// TIA Portal project "TIA_PP" (V19)

(* hardware
DEVICE "HMI_1"  KTP400 Basic PN
   slot 0: "HMI_1"  HMI  6AV2 123-2DB03-0AX0  13.0.1.0
   slot 1: "HMI_RT_1"  KTP400 Basic PN  6AV2 123-2DB03-0AX0  13.0.1.0
   slot 5: "HMI_1.IE_CP_1"  PROFINET Interface
      slot 1: "PROFINET Interface_1"  PROFINET Interface
         slot 1: "Port_1"  Port
DEVICE "S7-1200 station_1"  S7-1200 Station
   slot 0: "Rack_0"  Rack  V1.0
   slot 1: "PLC_1"  CPU 1212C AC/DC/Rly  6ES7 212-1BE40-0XB0  V4.1
*)

// ===== PLC "PLC_1"  CPU 1212C AC/DC/Rly =====

VAR_GLOBAL   // PLC tag table "Default tag table"
   "Tag_1" AT %MD5 : DWord;
   "Tag_2" AT %MD0 : DWord;
   "Tag_4" AT %MW5 : Word;
   "Tag_3" AT %MW10 : Int;
   "Tag_5" AT %M100.0 : Bool;
   "Warning light" AT %Q0.0 : Bool;
   "Tag_7" AT %M100.1 : Bool;
   "Motor1" AT %Q0.1 : Bool;
   "Tag_9" AT %MD5 : Time;
   "Tag_10" AT %MD12 : Real;
   "Tag_11" AT %MW15 : Int;
   "Tag_12" AT %ID30 : DWord;
   "Tag_13" AT %MD22 : Real;
   "Tag_14" AT %MW50 : Word;
   "LED" AT %Q0.2 : Bool;
   "Tag_16" AT %ID34 : DWord;
   "Tag_17" AT %MD25 : Real;
   "Tag_18" AT %MD26 : Real;
   "Fill Valve" AT %QD30 : Real;
   "Drain Valve" AT %QD34 : Real;
   "Tag_19" AT %M200.0 : Bool;
   "Tag_20" AT %M200.1 : Bool;
   "Animation bit" AT %M40.0 : Bool;
   "Clock_Byte" AT %MB300 : Byte;
   "Clock_10Hz" AT %M300.0 : Bool;
   "Clock_5Hz" AT %M300.1 : Bool;
   "Clock_2.5Hz" AT %M300.2 : Bool;
   "Clock_2Hz" AT %M300.3 : Bool;
   "Clock_1.25Hz" AT %M300.4 : Bool;
   "Clock_1Hz" AT %M300.5 : Bool;
   "Clock_0.625Hz" AT %M300.6 : Bool;
   "Clock_0.5Hz" AT %M300.7 : Bool;
   "Tag_21" AT %MB60 : Byte;
   "roller" AT %MD60 : Real;
   "roller_2" AT %MD70 : Real;
   "Tag_22" AT %MD65 : Real;
   "Tag_23" AT %MW60 : Int;
   "Tag_24" AT %MW65 : Int;
   "Down" AT %M90.0 : Bool;
   "Up" AT %M90.1 : Bool;
   "Tag_25" AT %MW75 : Int;
   "Tag_26" AT %MW78 : Int;
   "Tag_27" AT %MW80 : Int;
   "Alarm bit" AT %M99.0 : Bool;
   "Alarm register" AT %MW99 : Int;
   "OK bit" AT %M99.1 : Bool;
   "Reset Alarm" AT %M99.2 : Bool;
   "Start Button" AT %I0.0 : Bool;
   "Tag_28" AT %M0.1 : Bool;
   "Tag_6" AT %M0.2 : Bool;
   "Tag_15" AT %M0.3 : Bool;
   "Elpased time" AT %MD1 : Time;
   "Motor 2" AT %Q0.3 : Bool;
   "Tag_30" AT %Q0.4 : Bool;
   "LED1" AT %Q0.5 : Bool;
   "LED2" AT %Q0.6 : Bool;
   "Manual Button" AT %I0.5 : Bool;
   "Filling Button" AT %I0.6 : Bool;
   "Filling Value" AT %Q0.7 : Bool;
   "Draining Button" AT %I0.7 : Bool;
   "Draining Value" AT %Q1.0 : Bool;
   "Auto Button" AT %I0.1 : Bool;
   "Filling Button(1)" AT %I0.2 : Bool;
   "Tag_8" AT %M0.5 : Bool;
   "Tag_29" AT %M0.7 : Bool;
   "Tag_31" AT %M1.0 : Bool;
   "E-button" AT %M10.0 : Bool;
   "Stop Button" AT %M10.1 : Bool;
END_VAR

// folder: Basic Functions

DATA_BLOCK "PulseGenerator_DB"   // DB2
{ S7_Optimized_Access := 'TRUE' }
VERSION : 0.1
// stored: InstanceOfName PulseGenerator
"PulseGenerator"
BEGIN
END_DATA_BLOCK

DATA_BLOCK "ON-OFF Loop control_DB"   // DB3
{ S7_Optimized_Access := 'TRUE' }
VERSION : 0.1
// stored: InstanceOfName ON-OFF Loop control
"ON-OFF Loop control"
BEGIN
END_DATA_BLOCK

// folder: System blocks/Program resources

DATA_BLOCK "TP"   // DB1
{ S7_Optimized_Access := 'TRUE' }
AUTHOR : Simatic
FAMILY : IEC
NAME : IEC_TMR
VERSION : 1.0
// stored: InstanceOfName IEC_TIMER
"IEC_TIMER"
BEGIN
END_DATA_BLOCK

DATA_BLOCK "IEC_Timer_0_DB"   // DB4
{ S7_Optimized_Access := 'TRUE' }
AUTHOR : Simatic
FAMILY : IEC
NAME : IEC_TMR
VERSION : 1.0
// stored: InstanceOfName IEC_TIMER
"IEC_TIMER"
BEGIN
END_DATA_BLOCK

DATA_BLOCK "IEC_Timer_0_DB_1"   // DB5
{ S7_Optimized_Access := 'TRUE' }
AUTHOR : Simatic
FAMILY : IEC
NAME : IEC_TMR
VERSION : 1.0
// stored: InstanceOfName IEC_TIMER
"IEC_TIMER"
BEGIN
END_DATA_BLOCK

DATA_BLOCK "TON"   // DB6
{ S7_Optimized_Access := 'TRUE' }
AUTHOR : Simatic
FAMILY : IEC
NAME : IEC_TMR
VERSION : 1.0
// stored: InstanceOfName IEC_TIMER
"IEC_TIMER"
BEGIN
END_DATA_BLOCK

DATA_BLOCK "TOFF"   // DB7
{ S7_Optimized_Access := 'TRUE' }
AUTHOR : Simatic
FAMILY : IEC
NAME : IEC_TMR
VERSION : 1.0
// stored: InstanceOfName IEC_TIMER
"IEC_TIMER"
BEGIN
END_DATA_BLOCK

// folder: (top level)

FUNCTION "MHJ-PLC-Lab-Function-S71200" : Void   // FC1, SCL
{ S7_Optimized_Access := 'TRUE' }
VERSION : 0.1
   VAR_TEMP
      rdTimeReturn : Int;
      outputTime : DTL;
      SyncVal : Byte;
      forVal : Int;
      forVal_2 : Int;
      Value : Byte;
   END_VAR
   VAR CONSTANT
      CompVal : Byte := 16#34;
      Value_01 : Byte := 16#11;
      Value_01_DW : DWord := 16#A165_D992;
      Value_02_DW : DWord := 16#58BE_4401;
   END_VAR
BEGIN

   #Value := PEEK(area := 16#82,
                  dbNumber := 0,
                  byteOffset := 511);
   #Value := #Value + 1;

   POKE(area := 16#82,
        dbNumber := 0,
        byteOffset := 511,
        value := #Value);

   POKE(area := 16#81,
        dbNumber := 0,
        byteOffset := 1016,
        value := #Value_01_DW);
   POKE(area := 16#81,
        dbNumber := 0,
        byteOffset := 1020,
        value := #Value_02_DW);

   POKE(area := 16#81,
        dbNumber := 0,
        byteOffset := 511,
        value := B#16#00);

   FOR #forVal := 0 TO 120 DO
       FOR #forVal_2 := 0 TO 10 DO
           #rdTimeReturn := RD_SYS_T(#outputTime);
           #rdTimeReturn := WR_SYS_T(#outputTime);
           #rdTimeReturn := RD_SYS_T(#outputTime);
           #rdTimeReturn := WR_SYS_T(#outputTime);
       END_FOR;
       #SyncVal := PEEK(area := 16#81,
                        dbNumber := 0,
                        byteOffset := 511);
       IF #SyncVal = #CompVal THEN
           GOTO M_1;
       END_IF;
   END_FOR;
   RETURN;

   M_1:
   POKE(area := 16#81,
        dbNumber := 0,
        byteOffset := 511,
        value := B#16#0);
END_FUNCTION

ORGANIZATION_BLOCK "Main"   // OB1, LAD, ProgramCycle
TITLE = "Main Program Sweep (Cycle)"
{ S7_Optimized_Access := 'TRUE' }
VERSION : 0.1
   VAR_INPUT
      Initial_Call : Bool;   // Initial call of this OB
      Remanence : Bool;   // =True, if remanent data are available
   END_VAR
BEGIN

REGION Network 1
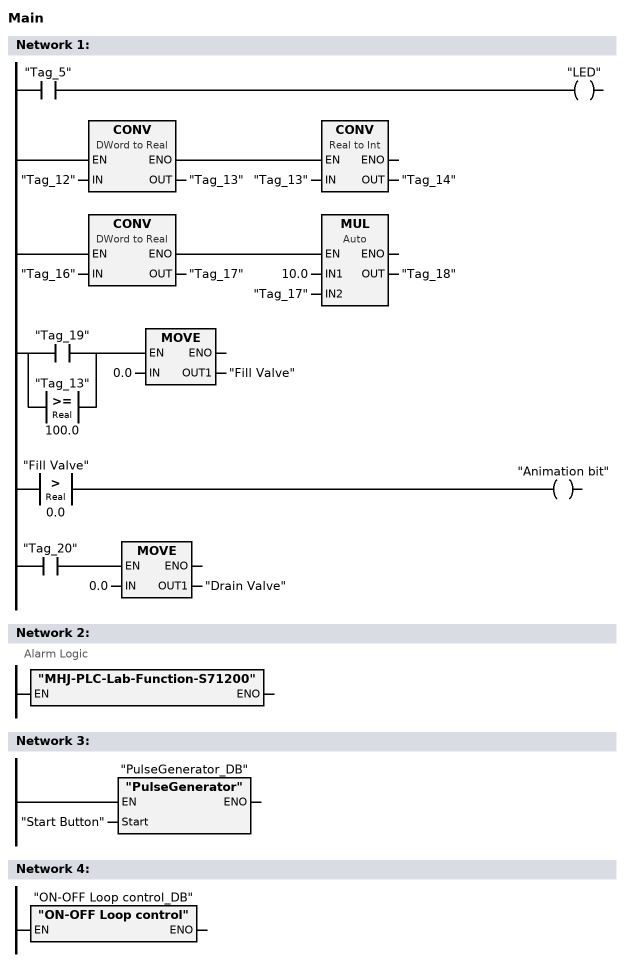
   // ENO of a box is taken as its EN; it also drops when the box reports an error
   "LED" := "Tag_5";
   "Tag_13" := DWORD_TO_REAL("Tag_12");
   "Tag_14" := REAL_TO_INT("Tag_13");
   "Tag_17" := DWORD_TO_REAL("Tag_16");
   "Tag_18" := 10.0 * "Tag_17";
   IF ("Tag_13" >= 100.0) OR "Tag_19" THEN "Fill Valve" := 0.0; END_IF;
   "Animation bit" := "Fill Valve" > 0.0;
   IF "Tag_20" THEN "Drain Valve" := 0.0; END_IF;
END_REGION

REGION Network 2
   // Alarm Logic
   RUNG wire#powerrail
      "MHJ-PLC-Lab-Function-S71200"()
   END_RUNG
   // the same network as SCL:
   "MHJ-PLC-Lab-Function-S71200"();
END_REGION

REGION Network 3
   RUNG wire#powerrail
      "PulseGenerator_DB"(Start := "Start Button")
   END_RUNG
   // the same network as SCL:
   "PulseGenerator_DB"(Start := "Start Button");   // "PulseGenerator"
END_REGION

REGION Network 4
   RUNG wire#powerrail
      "ON-OFF Loop control_DB"()
   END_RUNG
   // the same network as SCL:
   "ON-OFF Loop control_DB"();   // "ON-OFF Loop control"
END_REGION
END_ORGANIZATION_BLOCK

// folder: Basic Functions

FUNCTION_BLOCK "PulseGenerator"   // FB1, LAD
{ S7_Optimized_Access := 'TRUE' }
VERSION : 0.1
   VAR_INPUT
      Start : Bool;
   END_VAR
   VAR_TEMP   // added for the SCL form of the ladder/FBD networks
      _w1 : Bool;
      _w2 : Bool;
      _w3 : Bool;
   END_VAR
BEGIN

REGION Network 1: Pulse Generator
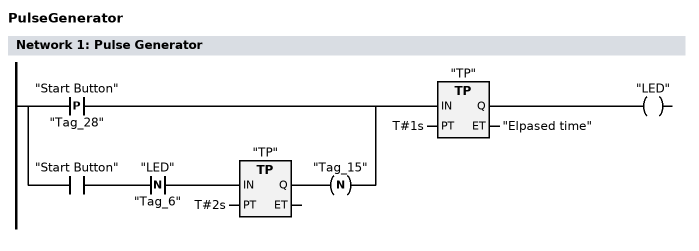
   #_w1 := "Start Button" AND NOT "Tag_28";   // rising edge of "Start Button"
   "Tag_28" := "Start Button";
   #_w2 := "Start Button" AND NOT "LED" AND "Tag_6";   // falling edge of "LED"
   "Tag_6" := "LED";
   "TP".TP(IN := #_w2, PT := T#2s);
   #_w3 := NOT "TP".Q AND "Tag_15";   // falling edge
   "Tag_15" := "TP".Q;
   "TP".TP(IN := #_w1 OR #_w3, PT := T#1s, ET => "Elpased time");
   "LED" := "TP".Q;
END_REGION
END_FUNCTION_BLOCK

FUNCTION_BLOCK "ON-OFF Loop control"   // FB2, LAD
{ S7_Optimized_Access := 'TRUE' }
VERSION : 0.1
   VAR_TEMP   // added for the SCL form of the ladder/FBD networks
      _w1 : Bool;
      _w2 : Bool;
      _w3 : Bool;
   END_VAR
BEGIN

REGION Network 1
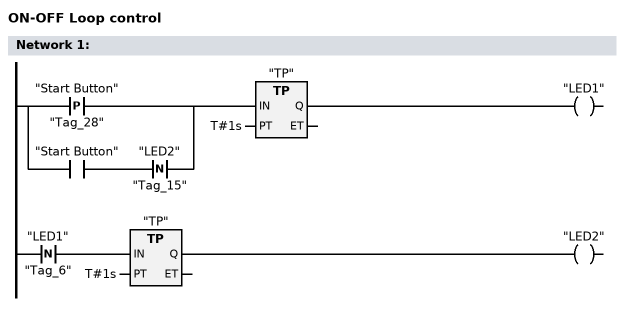
   #_w1 := "Start Button" AND NOT "Tag_28";   // rising edge of "Start Button"
   "Tag_28" := "Start Button";
   #_w2 := "Start Button" AND NOT "LED2" AND "Tag_15";   // falling edge of "LED2"
   "Tag_15" := "LED2";
   "TP".TP(IN := #_w1 OR #_w2, PT := T#1s);
   "LED1" := "TP".Q;
   #_w3 := NOT "LED1" AND "Tag_6";   // falling edge of "LED1"
   "Tag_6" := "LED1";
   "TP".TP(IN := #_w3, PT := T#1s);
   "LED2" := "TP".Q;
END_REGION
END_FUNCTION_BLOCK

FUNCTION_BLOCK "TimeON & OFF delay"   // FB3, LAD
{ S7_Optimized_Access := 'TRUE' }
VERSION : 0.1
BEGIN

REGION Network 1
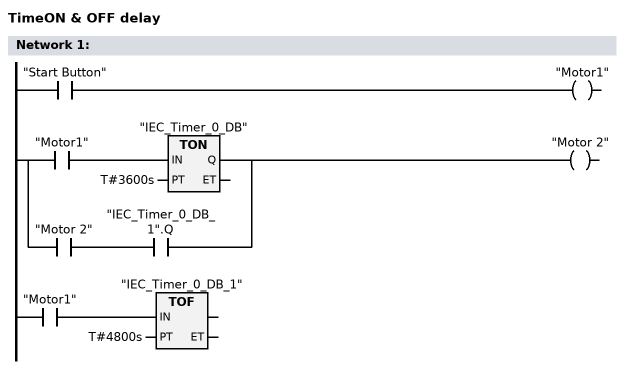
   "Motor1" := "Start Button";
   "IEC_Timer_0_DB".TON(IN := "Motor1", PT := T#3600s);
   "Motor 2" := "IEC_Timer_0_DB".Q OR ("Motor 2" AND "IEC_Timer_0_DB_1".Q);
   "IEC_Timer_0_DB_1".TOF(IN := "Motor1", PT := T#4800s);
END_REGION
END_FUNCTION_BLOCK

FUNCTION_BLOCK "TON_OFF value control"   // FB4, LAD
{ S7_Optimized_Access := 'TRUE' }
VERSION : 0.1
   VAR_TEMP   // added for the SCL form of the ladder/FBD networks
      _w1 : Bool;
      _w2 : Bool;
      _w3 : Bool;
      _w4 : Bool;
   END_VAR
BEGIN

REGION Network 1
   // Manual Mode ON - OFF
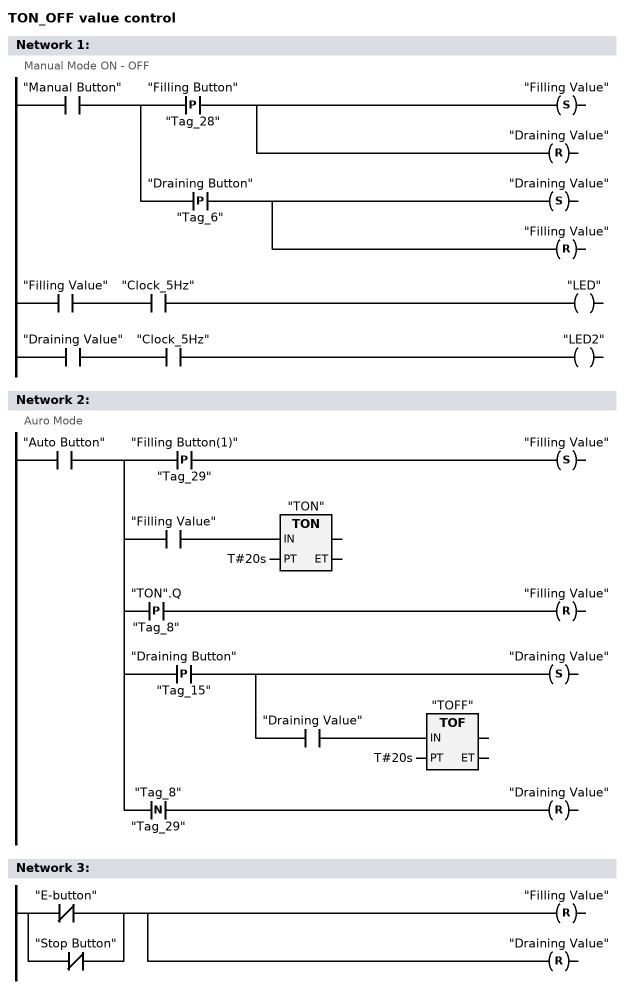
   RUNG wire#powerrail
      Contact( "Manual Button" )
      wire#w1
      P_Contact(operand := "Filling Button", bit := "Tag_28")
      wire#w2
      S_Coil( "Filling Value" )
   END_RUNG
   RUNG wire#w2
      R_Coil( "Draining Value" )
   END_RUNG
   RUNG wire#w1
      P_Contact(operand := "Draining Button", bit := "Tag_6")
      wire#w3
      S_Coil( "Draining Value" )
   END_RUNG
   RUNG wire#w3
      R_Coil( "Filling Value" )
   END_RUNG
   RUNG wire#powerrail
      Contact( "Filling Value" )
      Contact( "Clock_5Hz" )
      Coil( "LED" )
   END_RUNG
   RUNG wire#powerrail
      Contact( "Draining Value" )
      Contact( "Clock_5Hz" )
      Coil( "LED2" )
   END_RUNG
   // the same network as SCL:
   #_w1 := "Manual Button" AND "Filling Button" AND NOT "Tag_28";   // rising edge of "Filling Button"
   "Tag_28" := "Filling Button";
   IF #_w1 THEN
       "Filling Value" := TRUE;
       "Draining Value" := FALSE;
   END_IF;
   #_w2 := "Manual Button" AND "Draining Button" AND NOT "Tag_6";   // rising edge of "Draining Button"
   "Tag_6" := "Draining Button";
   IF #_w2 THEN
       "Draining Value" := TRUE;
       "Filling Value" := FALSE;
   END_IF;
   "LED" := "Filling Value" AND "Clock_5Hz";
   "LED2" := "Draining Value" AND "Clock_5Hz";
END_REGION

REGION Network 2
   // Auro Mode
   #_w1 := "Auto Button" AND "Filling Button(1)" AND NOT "Tag_29";   // rising edge of "Filling Button(1)"
   "Tag_29" := "Filling Button(1)";
   IF #_w1 THEN "Filling Value" := TRUE; END_IF;
   "TON".TON(IN := "Auto Button" AND "Filling Value", PT := T#20s);
   #_w2 := "Auto Button" AND "TON".Q AND NOT "Tag_8";   // rising edge of "TON".Q
   "Tag_8" := "TON".Q;
   IF #_w2 THEN "Filling Value" := FALSE; END_IF;
   #_w3 := "Auto Button" AND "Draining Button" AND NOT "Tag_15";   // rising edge of "Draining Button"
   "Tag_15" := "Draining Button";
   IF #_w3 THEN "Draining Value" := TRUE; END_IF;
   "TOFF".TOF(IN := #_w3 AND "Draining Value", PT := T#20s);
   #_w4 := "Auto Button" AND NOT "Tag_8" AND "Tag_29";   // falling edge of "Tag_8"
   "Tag_29" := "Tag_8";
   IF #_w4 THEN "Draining Value" := FALSE; END_IF;
END_REGION

REGION Network 3
   RUNG wire#powerrail
      I_Contact( "E-button" )
      wire#w1
      R_Coil( "Filling Value" )
   END_RUNG
   RUNG wire#powerrail
      I_Contact( "Stop Button" )
   END_RUNG wire#w1
   RUNG wire#w1
      R_Coil( "Draining Value" )
   END_RUNG
   // the same network as SCL:
   IF NOT "E-button" OR NOT "Stop Button" THEN
       "Filling Value" := FALSE;
       "Draining Value" := FALSE;
   END_IF;
END_REGION
END_FUNCTION_BLOCK

(* ===== HMI "HMI_RT_1" =====
system functions are stored by id; their names below are inferred from use
connection "HMI_Connection_1": ETHERNET, SMART_S7_1200_OMS

HMI tags "Default tag table"
   "Tag_5" : Bool = PLC Tag_5 AT %M100.0, 100 ms
   "Tag_7" : Bool = PLC Tag_7 AT %M100.1, 100 ms
   "Tag_6" : Bool = PLC "Warning light" AT %Q0.0, 100 ms
   "Tag_10" : Real = PLC Tag_10 AT %MD12, 1 s
   "Tag_11" : Int = PLC Tag_11 AT %MW15, 1 s
   "Tag_14" : Word = PLC Tag_14 AT %MW50, 100 ms
   "Tag_17" : Real = PLC Tag_17 AT %MD25, 100 ms
   "Tag_18" : Real = PLC Tag_18 AT %MD26, 100 ms
   "Fill Valve" : Real = PLC "Fill Valve" AT %QD30, 100 ms
   "Drain Valve" : Real = PLC "Drain Valve" AT %QD34, 100 ms
   "Tag_19" : Bool = PLC Tag_19 AT %M200.0, 100 ms
   "Tag_20" : Bool = PLC Tag_20 AT %M200.1, 100 ms
   "Animation bit" : Bool = PLC "Animation bit" AT %M40.0, 1 s
   "Tag_13" : Real = PLC Tag_13 AT %MD22, 1 s
   "Tag_21" : Byte = PLC Tag_21 AT %MB60, 100 ms
   "roller_HMI" : Real = PLC roller AT %MD60, 100 ms
   "roller_2" : Real = PLC roller_2 AT %MD70, 100 ms
   "Tag_23" : Int = PLC Tag_23 AT %MW60, 100 ms
   "Tag_25" : Int = PLC Tag_25 AT %MW75, 100 ms
   "Up" : Bool = PLC Up AT %M90.1, 100 ms
   "Alarm bit" : Bool = PLC "Alarm bit" AT %M99.0, 1 s
   "Alarm register" : Int = PLC "Alarm register" AT %MW99, 1 s
   "Logging Tag" : Bool AT %DB1.DBX0.0

discrete alarms
   1: 'Valve malfunctioning!', class Warnings, trigger "Alarm register" bit 8
   2: 'Valve OK', class Warnings, trigger "Alarm register" bit 9

graphic list "Roller": 0..249 '1'; 250..499 '2'; 500..749 '3'; 750..1000 '4'

graphic list "Motor": 0 'Graphic_24'; 1 'Graphic_25'

graphic list "Arrow": 0 'Graphic_27'; 1 'Graphic_26'

graphic list "Valve": 0 'OFF'; 1..7 'Partially ON_1'; 8..10 'ON_1'

graphic list "Pipes": 0 'not flowing'; 1..7 'Partially flowing'; 8..10 'flowing'

screen "Root screen" 480x272, template "Template_1"
   Button "Button_6" at 204,137 size 122x32; TextOff 'Tank Animation'
      on Press: ActivateScreen("Tank", 0)
   TextField "Text field_1" at 76,96 size 375x34; Text 'Trend View and Data Logging'
   GraphicView "Graphic view_1" at 223,8 size 83x67; Picture "logo"
   TextField "Text field_2" at 98,76 size 336x27; Text 'Learn Siemens S7-1200 & KTP 400'

screen "Tank" 480x272
   Bar "Bar_1" at 254,76 size 120x139; MinimumValue 0; MaximumValue 100
      ProcessValue <- "Tag_18"
   TextField "Text field_2" at 248,1 size 135x23; Text 'Tank Animation'
   GraphicView "Graphic view_1" at 254,60 size 122x18; Picture "Graphic_1"
   GraphicView "Graphic view_2" at 253,213 size 123x28; Picture "Graphic_13"
   Button "Button_4" at 429,190 size 45x23; TextOff 'OFF'
      on Press: function_b14e0dd5("Tag_20", 0)
   IOField "I/O field_1" at 383,60 size 43x29; FormatPattern 99.9
      ProcessValue <- "Fill Valve"
   IOField "I/O field_2" at 383,187 size 43x29; FormatPattern 99.9
      ProcessValue <- "Drain Valve"
   Button "Button_3" at 429,63 size 45x23; TextOff 'OFF'
      on Press: function_b14e0dd5("Tag_19", 0)
   IOField "I/O field_3" at 378,133 size 43x18; FormatPattern 999.9
      ProcessValue <- "Tag_18"
   GraphicView "Graphic view_5" at 295,34 size 33x28; Picture "Graphic_18"
   GraphicIOField "Graphic I/O field_1" at 387,27 size 39x32; PictureList "Valve"
      ProcessValue <- "Fill Valve"
   GraphicIOField "Graphic I/O field_2" at 385,230 size 39x32; PictureList "Valve"
      ProcessValue <- "Drain Valve"
   GraphicIOField "Graphic I/O field_3" at 327,41 size 62x13; PictureList "Pipes"
      ProcessValue <- "Fill Valve"
   GraphicIOField "Graphic I/O field_4" at 424,41 size 56x13; PictureList "Pipes"
      ProcessValue <- "Fill Valve"
   GraphicIOField "Graphic I/O field_5" at 325,245 size 62x13; PictureList "Pipes"
      ProcessValue <- "Drain Valve"
   GraphicIOField "Graphic I/O field_6" at 422,245 size 58x13; PictureList "Pipes"
      ProcessValue <- "Drain Valve"
   Rectangle "Rectangle_8" at 306,85 size 12x122
      Appearance <- "Fill Valve"
      Visibility <- "Animation bit"
   TextField "Text field_3" at 422,132 size 23x22; Text '%'
   GraphicView "Graphic view_3" at 303,239 size 23x25; Picture "Graphic_19"
   Button "Button_1" at 427,3 size 50x32; TextOff 'Home'
      on Press: ActivateScreen("Root screen", 0)
   TrendView "Trend view_1" at 3,5 size 250x201
   Button "Button_2" at 5,213 size 96x32; TextOff 'Start Logging'
      on Press: function_fd9437ed(0, "Tank Level"); SetBit("Logging Tag")
   Button "Button_5" at 106,214 size 96x30; TextOff 'Stop Logging'
      on Press: function_b6526003(0, "Tank Level"); ResetBit("Logging Tag")
   Button "Button_6" at 205,215 size 47x30; TextOff 'Clear'
      on Press: function_ff1151d2(0, "Tank Level")
   Rectangle "Rectangle_1" at 111,248 size 17x16
      Appearance <- "Logging Tag"
   TextField "Text field_1" at 6,246 size 102x20; Text 'Logging Status'

Template "Template_1" 480x272
   Button "Template_Button" at 388,227 size 63x44; TextOff 'ExitRuntime'; PictureOff "ExitRuntime_KTP400_Basic_PN_TR"; PictureOn "ExitRuntime_KTP400_Basic_PN_TR"
      on Release: StopRuntime(0)
   Button "Template_Button_3" at 28,227 size 63x44; TextOff 'NavigateHome'; PictureOff "NavigateHome_KTP400_Basic_PN_TR"; PictureOn "NavigateHome_KTP400_Basic_PN_TR"
      on Release: ActivateScreen("Root screen", 0)
*)